SUBAPPLICATION Uebung_003a2b_AX (* 2x R_IO mit IXA *)
  (* Standard: 61499-2; Description: Copyright (c) 2023 Meisterschulen am Ostbahnhof This program and the accompanying materials are made available under the terms of the Eclipse Public License 2.0 which is available at https://www.eclipse.org/legal/epl-2.0/ SPDX-License-Identifier: EPL-2.0 *)
  (* Version 1.0, 2026-01-13, Franz Höpfinger, Meisterschulen am Ostbahnhof, initial API and implementation and/or initial documentation *)
  PACKAGE Uebungen;
  IMPORT logiBUS::io::DI::logiBUS_DI::Input_I1;
  IMPORT logiBUS::io::DI::logiBUS_DI::Input_I2;
  IMPORT logiBUS::io::DI::logiBUS_DI::Input_I3;
  IMPORT logiBUS::io::DQ::logiBUS_DO::Output_Q1;
  IMPORT logiBUS::io::DQ::logiBUS_DO::Output_Q2;
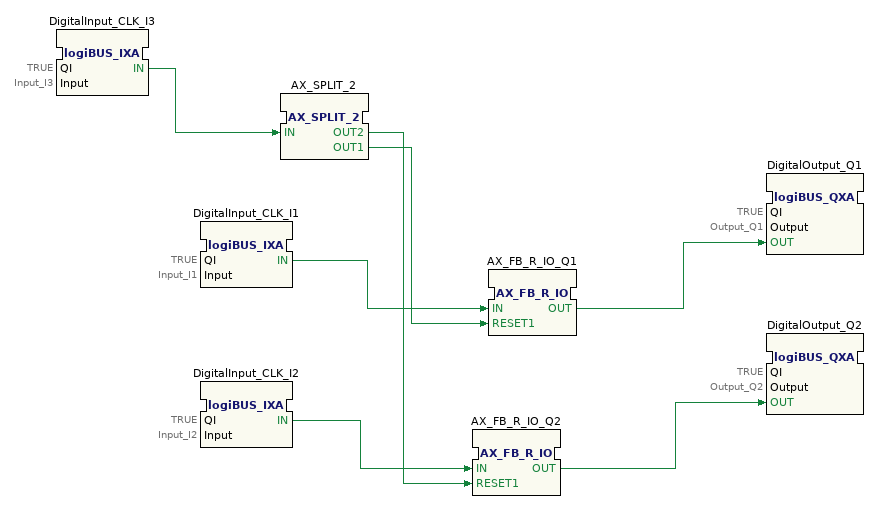
  (* Hausmeister-Aus (alles Aus mit einem Schalter) Schalter müsste RASTEND sein. Ansonsten ist nur solange aus wie der Taster gehalten wird. *)
  FBS
    DigitalOutput_Q1 : logiBUS::io::DQ::logiBUS_QXA(QI := TRUE, Output := Output_Q1);
    DigitalInput_CLK_I1 : logiBUS::io::DI::logiBUS_IXA(QI := TRUE, Input := Input_I1);
    DigitalInput_CLK_I2 : logiBUS::io::DI::logiBUS_IXA(QI := TRUE, Input := Input_I2);
    AX_FB_R_IO_Q1 : adapter::monostableElements::AX_FB_R_IO;
    DigitalInput_CLK_I3 : logiBUS::io::DI::logiBUS_IXA(QI := TRUE, Input := Input_I3);
    AX_FB_R_IO_Q2 : adapter::monostableElements::AX_FB_R_IO;
    DigitalOutput_Q2 : logiBUS::io::DQ::logiBUS_QXA(QI := TRUE, Output := Output_Q2);
    AX_SPLIT_2 : adapter::events::unidirectional::AX_SPLIT_2;
  END_FBS
  ADAPTER_CONNECTIONS
    AX_FB_R_IO_Q1.OUT TO DigitalOutput_Q1.OUT;
    AX_FB_R_IO_Q2.OUT TO DigitalOutput_Q2.OUT;
    DigitalInput_CLK_I1.IN TO AX_FB_R_IO_Q1.IN;
    DigitalInput_CLK_I2.IN TO AX_FB_R_IO_Q2.IN;
    DigitalInput_CLK_I3.IN TO AX_SPLIT_2.IN;
    AX_SPLIT_2.OUT2 TO AX_FB_R_IO_Q2.RESET1;
    AX_SPLIT_2.OUT1 TO AX_FB_R_IO_Q1.RESET1;
  END_CONNECTIONS
END_SUBAPPLICATION
